// TwinCAT 3 PLC project Device3
// ProgramVersion: 3.1.4026.20
// libraries:
//   Tc2_Standard, * (Beckhoff Automation GmbH)
//   Tc2_System, * (Beckhoff Automation GmbH)
// project tree:
//   GVLs/ GVL.TcGVL
//   / PlcTask.TcTTO
//   POUs/ MAIN.TcPOU
// real-time tasks:
//   TASK PlcTask: cycle T#10ms, priority 20, ADS port 350
//   TASK PlcTask1: cycle T#10ms, priority 21, ADS port 351

CONFIGURATION Device3
    RESOURCE PLC ON TwinCAT3
        TASK PlcTask(INTERVAL := T#10ms, PRIORITY := 21);
        PROGRAM MAIN WITH PlcTask : MAIN;
    END_RESOURCE
END_CONFIGURATION

// ---- GVLs/GVL.TcGVL
{attribute 'qualified_only'}
VAR_GLOBAL
    mb_Input_Coils 				: ARRAY [0..255] OF BOOL;
    mb_Output_Coils 			: ARRAY [0..255] OF BOOL;
    mb_Output_Registers 		: ARRAY [0..255] OF WORD;
    mb_Input_Registers 			: ARRAY [0..255] OF WORD;
END_VAR

// ---- POUs/MAIN.TcPOU
PROGRAM MAIN
VAR
    level : WORD := 0;
    pump : BOOL := FALSE;
    low : BOOL;
    high : BOOL;
    low_3 : INT := 0;
    high_3 : INT := 3;
END_VAR

level := GVL.mb_Output_Registers[0];

low := level <=  low_3;
high := level >= high_3;
pump := NOT(low) AND (high OR pump);

GVL.mb_Input_Coils[0] := pump;

END_PROGRAM
